INTERFACE I_PiezoDrive

METHOD Brake : BOOL
VAR_INPUT
END_VAR
END_METHOD

METHOD Halt : BOOL
VAR_INPUT
END_VAR
END_METHOD

METHOD Home : BOOL
VAR_INPUT
END_VAR
END_METHOD

METHOD Interlock
VAR_INPUT
END_VAR
END_METHOD

METHOD Logger : BOOL
VAR_INPUT
END_VAR
END_METHOD

METHOD MoveAbsolute
VAR_INPUT
END_VAR
END_METHOD

METHOD MoveVelocity
VAR_INPUT
END_VAR
END_METHOD

METHOD Power : BOOL
VAR_INPUT
END_VAR
END_METHOD

METHOD Reset : BOOL
VAR_INPUT
END_VAR
END_METHOD

END_INTERFACE

(* stored: Version 1.1.0.1
   Itf I_PiezoDrive: Id {49729736-8717-4a13-800f-a53162ccda84}
   Method Brake: Id {e0529470-e1a2-408b-acaa-cacbe414aa6e}
   Method Halt: Id {1645d0ef-eb4b-4235-b6cc-4a214463d443}
   Method Home: Id {f7b9941e-fd39-45a3-99c7-fc867c3625ba}
   Method Interlock: Id {b9614087-83f0-4675-8dad-b6765017e9ea}
   Method Logger: Id {36d29a03-8107-42f2-b596-87523b11c29f}
   Method MoveAbsolute: Id {c32a9e13-f332-4841-9fc3-9751e2083446}
   Method MoveVelocity: Id {bc7db01d-6c11-4d35-a626-79d63771cf0a}
   Method Power: Id {08548eb9-8f7d-4758-8069-c44e4c6df0ba}
   Method Reset: Id {43fc3192-2758-4d04-872e-08906cd5bf28} *)
